INTERFACE ITF_Cyclic

METHOD Cycle : BOOL
VAR_INPUT
END_VAR
END_METHOD

END_INTERFACE

(* stored: Version 1.1.0.1, ProductVersion 3.1.4024.12
   Itf ITF_Cyclic: Id {e211f975-93c3-4743-b545-3e91459af86e}
   Method Cycle: Id {ce275aa3-f435-460f-965e-310d808f2565} *)
